(* Copyright 2017 Cimpress

Licensed under the Apache License, Version 2.0 (the "License");
you may not use this file except in compliance with the License.
You may obtain a copy of the License at

http://www.apache.org/licenses/LICENSE-2.0

Unless required by applicable law or agreed to in writing, software
distributed under the License is distributed on an "AS IS" BASIS,
WITHOUT WARRANTIES OR CONDITIONS OF ANY KIND, either express or implied.
See the License for the specific language governing permissions and
limitations under the License. *)

TYPE T_Ctrl_IoUsint :
STRUCT
	///mapped io variable to hardware
	map: USINT;
	///shows the state of (input: mapped, output: set by programm respectiv at the moment one cycle later evtl. from the forcing if forcing active) -> necessary for what?
	state: USINT;
	///variabel to/ from program
	intern: USINT;
	///variabel set from UI
	force: USINT;
	///enable force of single io-datapoint
	EnForce: BOOL;
END_STRUCT
END_TYPE

(* stored: Version 1.1.0.1, ProductVersion 3.1.4019.2
   DUT T_Ctrl_IoUsint: Id {1206ecb9-8ab9-4733-859a-9fb1e8d36978} *)
